// Mitsubishi GX Works2 project: a11   PLC: Q02/Q02H

PROGRAM MAIN
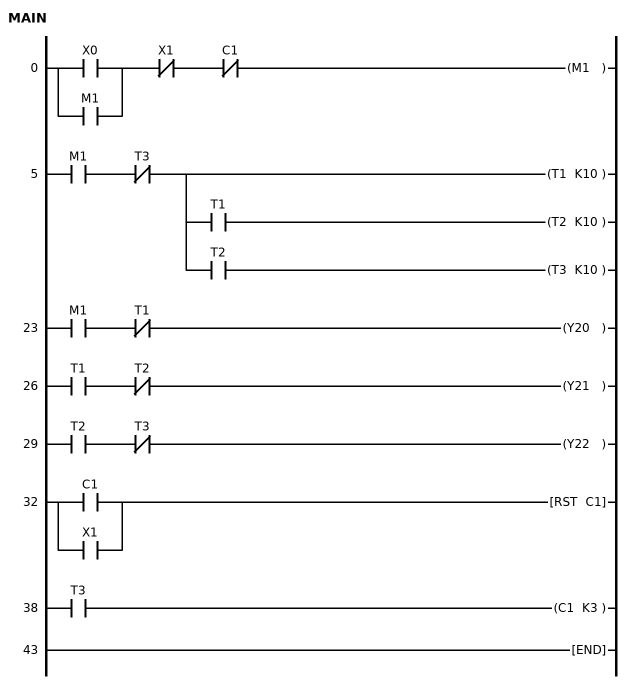
0     LD      X0
      OR      M1
      ANI     X1
      ANI     C1
      OUT     M1
5     LD      M1
      ANI     T3
      OUT     T1 K10
      MPS
      AND     T1
      OUT     T2 K10
      MPP
      AND     T2
      OUT     T3 K10
23    LD      M1
      ANI     T1
      OUT     Y20
26    LD      T1
      ANI     T2
      OUT     Y21
29    LD      T2
      ANI     T3
      OUT     Y22
32    LD      C1
      OR      X1
      RST     C1
38    LD      T3
      OUT     C1 K3
43    END
END_PROGRAM
